# EPICS substitutions: modules/event/evrSupport/Db/ioc/IOC-IN20-LS11bsa.substitutions
#
# BSA records

file bsaPWREdef.db {
#          Device        ,loc'n , IOC unit, timing system
  pattern {    DEVICE    , LOC  ,  UN , SLCLNK                  }
	  { LASR:IN20:156, IN20 , LS11, ""                      }
	  { LASR:IN20:196, IN20 , LS11, ""                      }
}
